FUNCTION_BLOCK FB_CRYO_VALVE_CTRL EXTENDS FB_CRYO_BIN_CTRL
VAR_INPUT
END_VAR
VAR_OUTPUT
END_VAR
VAR
END_VAR

// Execute parent FB.
SUPER^();

METHOD M_SetStatus
VAR_INPUT
	nState:	E_CRYO_BIN_CTRL_STATE;
END_VAR
// Execute the status of the parent FB
SUPER^.M_SetStatus(nState);

// Set proper error description, if any.
IF Actuator.stat.bError THEN
	stat.sState	:= 'Valve failure';
END_IF
END_METHOD

METHOD M_User_SetAction : INT
VAR_INPUT
END_VAR
// TODO USER
// Set Valve command based on the input parameter in_bEnable.
//
	
IF	stat.nState = E_CRYO_BIN_CTRL_STATE.ACTIVE_OFF  AND in_bEnable THEN
	// Activate the actuator, i.e. open the valve
	M_User_SetAction	:= E_CRYO_BIN_CTRL_ACTION.ON;
ELSIF  stat.nState = E_CRYO_BIN_CTRL_STATE.ACTIVE_ON AND NOT in_bEnable THEN
	// Dectivate the actuator, i.e. close the valve
	M_User_SetAction	:= E_CRYO_BIN_CTRL_ACTION.OFF;
ELSE
	// Don't do anything
	M_User_SetAction	:= E_CRYO_BIN_CTRL_ACTION.NONE;
END_IF
END_METHOD

END_FUNCTION_BLOCK

(* stored: Version 1.1.0.1, ProductVersion 3.1.4024.9
   POU FB_CRYO_VALVE_CTRL: Id {821ef5cb-5c3c-4548-8cdd-f457c89df676}, SpecialFunc None
   Method M_SetStatus: Id {4aedb583-a641-44e2-9926-6d1ee3abadf1}
   Method M_User_SetAction: Id {60abe389-4ad1-49f5-a9ed-250397cb9229} *)
